// TIA Portal V17 export
// export: Created 2023-12-22T15:08:09.508465Z, ExportSetting WithDefaults, DisplayName Totally Integrated Automation Portal, DisplayVersion V17, DisplayName TIA Portal Openness, DisplayVersion V17, DisplayName TIA Portal Version Control Interface, DisplayVersion V17, DisplayName STEP 7 Professional, DisplayVersion V17, DisplayName STEP 7 Safety, DisplayVersion V17, DisplayName WinCC Advanced, DisplayVersion V17
DATA_BLOCK "ModBus_TCP_DB"   // DB40
VERSION : 0.1
// stored: AutoNumber false, DBAccessibleFromOPCUA true, DBAccessibleFromWebserver true, InstanceOfName ModBus_TCP, InstanceOfType FB
"ModBus_TCP"
   // VAR RETAIN
   //    DATA : Array[0..100] of Word;
   //    "Step" : Int;
   //    Device : Int;
   //    Limit { S7_SetPoint := 'True'} : Int := 10;
   //    COM_Control : Struct
   //       Enable { S7_SetPoint := 'True'} : Bool := TRUE;
   //       Start : Bool;
   //       Reset : Bool;
   //       REQ_Done : Bool;
   //       REQ_Busy : Bool;
   //       REQ_Error : Bool;
   //       REQ_Status : Word;
   //       Error_Code : Word;
   //       Status : Int;
   //    END_STRUCT;
   //    COM_REQ : Struct
   //       ADDR : UInt;
   //       MODE : USInt;
   //       Register : UDInt;
   //       Length : UInt;
   //    END_STRUCT;
   //    CONNECT { S7_SetPoint := 'True'} : TCON_IP_v4;
   //    DEV_Config : Array[1..10] of Struct
   //       Use { S7_SetPoint := 'True'} : Bool;
   //       MODE { S7_SetPoint := 'True'} : Bool;
   //       ADDR { S7_SetPoint := 'True'} : UInt;
   //       Register { S7_SetPoint := 'True'} : UDInt;
   //       Length { S7_SetPoint := 'True'} : UInt;
   //       Source_DB { S7_SetPoint := 'True'} : UInt;
   //       Source_OFFSET { S7_SetPoint := 'True'} : UInt;
   //       Target_DB { S7_SetPoint := 'True'} : UInt;
   //       Target_OFFSET { S7_SetPoint := 'True'} : UInt;
   //       Status : UInt;
   //    END_STRUCT;
   //    MB_CLIENT : MB_CLIENT;
   //    T_Busy : "Time_M";
   // END_VAR
BEGIN
   CONNECT.InterfaceId := 64;
   CONNECT.ID := 1;
   CONNECT.ConnectionType := 11;
   CONNECT.RemoteAddress.ADDR[1] := 192;
   CONNECT.RemoteAddress.ADDR[2] := 168;
   CONNECT.RemoteAddress.ADDR[3] := 0;
   CONNECT.RemoteAddress.ADDR[4] := 10;
   CONNECT.RemotePort := 502;
   DEV_Config[1..10].Use := FALSE;
   DEV_Config[1..10].MODE := FALSE;
   DEV_Config[1..10].ADDR := 0;
   DEV_Config[1..10].Register := 0;
   DEV_Config[1..10].Length := 0;
   DEV_Config[1..10].Source_DB := 0;
   DEV_Config[1..10].Source_OFFSET := 0;
   DEV_Config[1..10].Target_DB := 0;
   DEV_Config[1..10].Target_OFFSET := 0;
END_DATA_BLOCK
